PROGRAM DBSync
VAR_INPUT
	bExportTrigger : BOOL ;
	bImportTrigger : BOOL ;
END_VAR
VAR
	Process : NT_StartProcess;

    bError : BOOL;
    iErrorId : UDINT;
	bIsBusy : BOOL;
END_VAR

IF bExportTrigger THEN
	Process(
    	NETID := '', 
    	PATHSTR := 'C:\Windows\System32\cmd.exe',  
		COMNDLINE := '/C start cmd /c C:\Users\Administrator\Documents\Scripts\Export.cmd',
		TMOUT := T#1M,
    	ERR => bError,            
    	ERRID => iErrorId,
		BUSY => bIsBusy       
	);
	
	
	Process(START:=TRUE);
    Process(START:=FALSE);
    bExportTrigger := FALSE;
	
ELSIF bImportTrigger THEN
	Process(
    	NETID := '', 
    	PATHSTR := 'C:\Windows\System32\cmd.exe',
    	COMNDLINE := '/C start cmd /c C:\Users\Administrator\Documents\Scripts\Import.cmd',      
    	ERR => bError,            
    	ERRID => iErrorId           
	);
    bImportTrigger := FALSE;
    Process(START:=TRUE);
    Process(START:=FALSE);
	
END_IF

END_PROGRAM

(* stored: Version 1.1.0.1, ProductVersion 3.1.4024.12
   POU DBSync: Id {c1e38521-1498-49b4-afde-113214ab9c62}, SpecialFunc None *)
